DATA_BLOCK "TRAVEL_PROFIBUS"	// DB 18
VERSION : 0.1
  STRUCT
   TRVLDRV1_REF_WITH_LIMIT : BOOL ;	//TRAVEL DRIVE-1 RESERVED1 BIT
   TRVLDRV1_LOCAL_REMOTE_BI : BOOL ;	//TRAVEL DRIVE-1 PROFIBUS SELECTED BIT
   TRVLDRV1_ACT_ABOVE_LMIT : BOOL ;	//TRAVEL DRIVE-1 REFERENCE REACHED BIT
   TRVLDRV1_PROFI_SELECTED : BOOL ;	//TRAVEL DRIVE-1 RESERVED2 BIT
   TRVLDRV1_EXTRNL_RUN_BIT : BOOL ;	//TRAVEL DRIVE-1 RESERVED3 BIT
   TRVLDRV1_RESERVED1_BIT : BOOL ;	//TRAVEL DRIVE-1 RESERVED4 BIT
   TRVLDRV1_RESERVED2_BIT : BOOL ;	//TRAVEL DRIVE-1 RESERVED5 BIT
   TRVLDRV1_RESERVED3_BIT : BOOL ;	//TRAVEL DRIVE-1 REVERSE DIRECTION BIT
   TRVLDRV1_RDY_SWITCH_ON : BOOL ;	//TRAVEL DRIVE-1 READY TO SWITCH ON BIT
   TRVLDRV1_RDY_BIT : BOOL ;	//TRAVEL DRIVE-1 READY BIT
   TRVLDRV1_RUNNING_BIT : BOOL ;	//TRAVEL DRIVE-1 RUNNING BIT
   TRVLDRV1_FAULT_BIT : BOOL ;	//TRAVEL DRIVE-1 FAULT BIT
   TRVLDRV1_OFF2_BIT : BOOL ;	//TRAVEL DRIVE-1 VOLTAGE ENABLED BIT
   TRVLDRV1_OFF3_BIT : BOOL ;	//TRAVEL DRIVE-1 EMERGENCY STOP BIT
   TRVLDRV1_SWTCHON_DISABLE : BOOL ;	//TRAVEL DRIVE-1 SWITCH ON DISABLE BIT
   TRVLDRV1_ALARM_BIT : BOOL ;	//TRAVEL DRIVE-1 ALARM BIT
   TRVLDRV1_SPEED_ACTUAL : INT ;	//TRAVEL DRIVE-1 SPEED ACTUAL VALUE
   TRAV_DRV_1_CURR_VAL : INT ;	//TRAVEL DRIVE 1 CURRENT VALUE
   TRV1_SPARE2_STATUS : WORD ;	//Temporary placeholder variable
   TRV1_SPARE3_STATUS : WORD ;	//Temporary placeholder variable
   TRV1_SPARE4_STATUS : WORD ;	//Temporary placeholder variable
   TRV1_SPARE5_STATUS : WORD ;	//Temporary placeholder variable
   TRV1_SPARE6_STATUS : WORD ;	//Temporary placeholder variable
   TRV1_SPARE7_STATUS : WORD ;	//Temporary placeholder variable
   TRV1_SPARE8_STATUS : WORD ;	//Temporary placeholder variable
   TRVLDRV1_CONTROLWORD : WORD ;	//TRAVEL DRIVE-1 CONTROL WORD VALUE
   TRVLDRV1_SPEED_REF : INT ;	//TRVVEL DRIVE-1 SPEED REFERENCE VALUE
   PZD3_DW1_3 : WORD ;	//PROCESS DATA FOR DRIVE
   TRV1_SPARE2_CNTL_WORD : WORD ;	//Temporary placeholder variable
   TRV1_SPARE3_CNTL_WORD : WORD ;	//Temporary placeholder variable
   TRV1_SPARE4_CNTL_WORD : WORD ;	//Temporary placeholder variable
   TRV1_SPARE5_CNTL_WORD : WORD ;	//Temporary placeholder variable
   TRV1_SPARE6_CNTL_WORD : WORD ;	//Temporary placeholder variable
   TRV1_SPARE7_CNTL_WORD : WORD ;	//Temporary placeholder variable
   TRV1_SPARE8_CNTL_WORD : WORD ;	//Temporary placeholder variable
   TRVLDRV2_REF_WITH_LIMIT : BOOL ;	//TRAVEL DRIVE-2 RESERVED1 BIT
   TRVLDRV2_LOCAL_REMOTE_BI : BOOL ;	//TRAVEL DRIVE-2 PROFIBUS SELECTED BIT
   TRVLDRV2_ACT_ABOVE_LMIT : BOOL ;	//TRAVEL DRIVE-2 REFERENCE REACHED BIT
   TRVLDRV2_PROFI_SELECTED : BOOL ;	//TRAVEL DRIVE-2 RESERVED2 BIT
   TRVLDRV2_EXTRNL_RUN_BIT : BOOL ;	//TRAVEL DRIVE-2 RESERVED3 BIT
   TRVLDRV2_RESERVED1_BIT : BOOL ;	//TRAVEL DRIVE-2 RESERVED4 BIT
   TRVLDRV2_RESERVED2_BIT : BOOL ;	//TRAVEL DRIVE-2 RESERVED5 BIT
   TRVLDRV2_RESERVED3_BIT : BOOL ;	//TRAVEL DRIVE-2 REVERSE DIRECTION BIT
   TRVLDRV2_RDY_SWITCH_ON : BOOL ;	//TRAVEL DRIVE-2 READY TO SWITCH ON BIT
   TRVLDRV2_RDY_BIT : BOOL ;	//TRAVEL DRIVE-2 READY BIT
   TRVLDRV2_RUNNING_BIT : BOOL ;	//TRAVEL DRIVE-2 RUNNING BIT
   TRVLDRV2_FAULT_BIT : BOOL ;	//TRAVEL DRIVE-2 FAULT BIT
   TRVLDRV2_OFF2_BIT : BOOL ;	//TRAVEL DRIVE-2 VOLTAGE ENABLED BIT
   TRVLDRV2_OFF3_BIT : BOOL ;	//TRAVEL DRIVE-2 EMERGENCY STOP BIT
   STAT_2 : BOOL ;	//TRAVEL DRIVE-2 SWITCH ON DISABLE BIT
   TRVLDRV2_ALARM_BIT : BOOL ;	//TRAVEL DRIVE-2 ALARM BIT
   TRVLDRV2_SPEED_ACTUAL : INT ;	//TRAVEL DRIVE-2 SPEED ACTUAL VALUE
   TRAV_DRV_2_CURR_VAL : INT ;	//TRAVEL DRIVE 2 CURRENT VALUE
   TRV2_SPARE2_STATUS : WORD ;	//Temporary placeholder variable
   TRV2_SPARE3_STATUS : WORD ;	//Temporary placeholder variable
   TRV2_SPARE4_STATUS : WORD ;	//Temporary placeholder variable
   TRV2_SPARE5_STATUS : WORD ;	//Temporary placeholder variable
   TRV2_SPARE6_STATUS : WORD ;	//Temporary placeholder variable
   TRV2_SPARE7_STATUS : WORD ;	//Temporary placeholder variable
   TRV2_SPARE8_STATUS : WORD ;	//Temporary placeholder variable
   TRVLDRV2_CONTROLWORD : WORD ;	//TRAVEL DRIVE-2 CONTROL WORD VALUE
   TRVLDRV2_SPEED_REF : INT ;	//TRVVEL DRIVE-2 SPEED REFERENCE VALUE
   TRVLDRV2_REF_2 : WORD ;	//TRAVEL DRIVE-2 SPEED REFERENCE VALUE
   AUX_DS_REF3 : WORD ;	//AUXILLIARY DATA SET REF 3
   TRV2_SPARE3_CNTL_WORD : WORD ;	//Temporary placeholder variable
   TRV2_SPARE4_CNTL_WORD : WORD ;	//Temporary placeholder variable
   TRV2_SPARE5_CNTL_WORD : WORD ;	//Temporary placeholder variable
   TRV2_SPARE6_CNTL_WORD : WORD ;	//Temporary placeholder variable
   TRV2_SPARE7_CNTL_WORD : WORD ;	//Temporary placeholder variable
   TRV2_SPARE8_CNTL_WORD : WORD ;	//Temporary placeholder variable
  END_STRUCT ;	
BEGIN
END_DATA_BLOCK

DATA_BLOCK "SF_PROFIBUS"	// DB 19
VERSION : 0.1
  STRUCT
   SF1_REF_WITH_LIMIT : BOOL ;	//SCREW FEEDER DRIVE-1 RESERVED1 BIT
   SF1_LOCAL_REMOTE_BI : BOOL ;	//SCREW FEEDER DRIVE-1 PROFIBUS SELECTED BIT
   SF1_ACT_ABOVE_LMIT : BOOL ;	//SCREW FEEDER DRIVE-1 REFERENCE REACHED BIT
   SF1_PROFI_SELECTED : BOOL ;	//SCREW FEEDER DRIVE-1 RESERVED2 BIT
   SF1_EXTRNL_RUN_BIT : BOOL ;	//SCREW FEEDER DRIVE-1 RESERVED3 BIT
   SF1_RESERVED1_BIT : BOOL ;	//SCREW FEEDER DRIVE-1 RESERVED4 BIT
   SF1_RESERVED2_BIT : BOOL ;	//SCREW FEEDER DRIVE-1 RESERVED5 BIT
   SF1_RESERVED3_BIT : BOOL ;	//SCREW FEEDER DRIVE-1 REVERSE DIRECTION BIT
   SF1_RDY_SWITCH_ON : BOOL ;	//SCREW FEEDER DRIVE-1 READY TO SWITCH ON BIT
   SF1_RDY_BIT : BOOL ;	//SCREW FEEDER DRIVE-1 READY BIT
   SF1_RUNNING_BIT : BOOL ;	//SCREW FEEDER DRIVE-1 RUNNING BIT
   SF1_FAULT_BIT : BOOL ;	//SCREW FEEDER DRIVE-1 FAULT BIT
   SF1_OFF2_BIT : BOOL ;	//SCREW FEEDER DRIVE-1 VOLTAGE ENABLED BIT
   SF1_OFF3_BIT : BOOL ;	//SCREW FEEDER DRIVE-1 EMERGENCY STOP BIT
   SF1_SWTCHON_DISABLE : BOOL ;	//SCREW FEEDER DRIVE-1 SWITCH ON DISABLE BIT
   SF1_ALARM_BIT : BOOL ;	//SCREW FEEDER DRIVE-1 ALARM BIT
   SF1_SPEED_ACTUAL : INT ;	//SCREW FEEDER DRIVE-1 SPEED ACTUAL VALUE
   SF_1_CURR_VAL : INT ;	//SCREW FEEDER DRIVE-1 CURRENT VALUE
   SF1_SPARE2_STATUS : WORD ;	//SCREW FEEDER SPARE STATUS WORD
   SF1_SPARE3_STATUS : WORD ;	//SCREW FEEDER SPARE STATUS WORD
   SF1_SPARE4_STATUS : WORD ;	//SCREW FEEDER SPARE STATUS WORD
   SF1_SPARE5_STATUS : WORD ;	//SCREW FEEDER SPARE STATUS WORD
   SF1_SPARE6_STATUS : WORD ;	//SCREW FEEDER SPARE STATUS WORD
   SF1_SPARE7_STATUS : WORD ;	//SCREW FEEDER SPARE STATUS WORD
   SF1_SPARE8_STATUS : WORD ;	//SCREW FEEDER SPARE STATUS WORD
   SF1_CONTROLWORD : WORD ;	//SCREW FEEDER DRIVE-1 CONTROL WORD VALUE
   SF1_SPEED_REF : INT ;	//SCREW FEEDER DRIVE-1 SPEED REFERENCE VALUE
   SF1_SPARE1_CNTL_WORD : WORD ;	//SCREW FEEDER SPARE CONTROL WORD
   SF1_SPARE2_CNTL_WORD : WORD ;	//SCREW FEEDER SPARE CONTROL WORD
   SF1_SPARE3_CNTL_WORD : WORD ;	//SCREW FEEDER SPARE CONTROL WORD
   SF1_SPARE4_CNTL_WORD : WORD ;	//SCREW FEEDER SPARE CONTROL WORD
   SF1_SPARE5_CNTL_WORD : WORD ;	//SCREW FEEDER SPARE CONTROL WORD
   SF1_SPARE6_CNTL_WORD : WORD ;	//SCREW FEEDER SPARE CONTROL WORD
   SF1_SPARE7_CNTL_WORD : WORD ;	//SCREW FEEDER SPARE CONTROL WORD
   SF1_SPARE8_CNTL_WORD : WORD ;	//SCREW FEEDER SPARE CONTROL WORD
   SF2_REF_WITH_LIMIT : BOOL ;	//SCREW FEEDER DRIVE-2 RESERVED1 BIT
   SF2_LOCAL_REMOTE_BIT : BOOL ;	//SCREW FEEDER DRIVE-2 PROFIBUS SELECTED BIT
   SF2_ACT_ABOVE_LMIT : BOOL ;	//SCREW FEEDER DRIVE-2 REFERENCE REACHED BIT
   SF2_PROFI_SELECTED : BOOL ;	//SCREW FEEDER DRIVE-2 RESERVED2 BIT
   SF2_EXTRNL_RUN_BIT : BOOL ;	//SCREW FEEDER DRIVE-2 RESERVED3 BIT
   SF2_RESERVED1_BIT1 : BOOL ;	//SCREW FEEDER DRIVE-2 RESERVED4 BIT
   SF2_RESERVED2_BIT : BOOL ;	//SCREW FEEDER DRIVE-2 RESERVED5 BIT
   SF2_RESERVED3_BIT : BOOL ;	//SCREW FEEDER DRIVE-2 REVERSE DIRECTION BIT
   SF2_RDY_SWITCH_ON : BOOL ;	//SCREW FEEDER DRIVE-2 READY TO SWITCH ON BIT
   SF2_RDY_BIT : BOOL ;	//SCREW FEEDER DRIVE-2 READY BIT
   SF2_RUNNING_BIT : BOOL ;	//SCREW FEEDER DRIVE-2 RUNNING BIT
   SF2_FAULT_BIT : BOOL ;	//SCREW FEEDER DRIVE-2 FAULT BIT
   SF2_OFF2_BIT : BOOL ;	//SCREW FEEDER DRIVE-2 VOLTAGE ENABLED BIT
   SF2_OFF3_BIT : BOOL ;	//SCREW FEEDER DRIVE-2 EMERGENCY STOP BIT
   SF2_SWTCHON_DISABLE : BOOL ;	//SCREW FEEDER DRIVE-2 SWITCH ON DISABLE BIT
   SF2_ALARM_BIT : BOOL ;	//SCREW FEEDER DRIVE-2 ALARM BIT
   SF2_SPEED_ACTUAL : INT ;	//SCREW FEEDER DRIVE-2 SPEED ACTUAL VALUE
   SF_2_CURR_VAL : INT ;	//SCREW FEEDER DRIVE 2 CURRENT VALUE
   SF2_SPARE2_STATUS : WORD ;	//SCREW FEEDER SPARE STATUS WORD
   SF2_SPARE3_STATUS : WORD ;	//SCREW FEEDER SPARE STATUS WORD
   SF2_SPARE4_STATUS : WORD ;	//SCREW FEEDER SPARE STATUS WORD
   SF2_SPARE5_STATUS : WORD ;	//SCREW FEEDER SPARE STATUS WORD
   SF2_SPARE6_STATUS : WORD ;	//SCREW FEEDER SPARE STATUS WORD
   SF2_SPARE7_STATUS : WORD ;	//SCREW FEEDER SPARE STATUS WORD
   SF2_SPARE8_STATUS : WORD ;	//SCREW FEEDER SPARE STATUS WORD
   SF2_CONTROLWORD : WORD ;	//SCREW FEEDER DRIVE-2 CONTROL WORD VALUE
   SF2_SPEED_REF : INT ;	//SCREW FEEDER DRIVE-2 SPEED REFERENCE VALUE
   SF2_SPARE1_CNTL_WORD : WORD ;	//SCREW FEEDER SPARE CONTROL WORD
   SF2_SPARE2_CNTL_WORD : WORD ;	//SCREW FEEDER SPARE CONTROL WORD
   SF2_SPARE3_CNTL_WORD : WORD ;	//SCREW FEEDER SPARE CONTROL WORD
   SF2_SPARE4_CNTL_WORD : WORD ;	//SCREW FEEDER SPARE CONTROL WORD
   SF2_SPARE5_CNTL_WORD : WORD ;	//SCREW FEEDER SPARE CONTROL WORD
   SF2_SPARE6_CNTL_WORD : WORD ;	//SCREW FEEDER SPARE CONTROL WORD
   SF2_SPARE7_CNTL_WORD : WORD ;	//SCREW FEEDER SPARE CONTROL WORD
   SF2_SPARE8_CNTL_WORD : WORD ;	//SCREW FEEDER SPARE CONTROL WORD
   SF3_REF_WITH_LIMIT : BOOL ;	//SCREW FEEDER DRIVE-3 RESERVED1 BIT
   SF3_LOCAL_REMOTE_BIT : BOOL ;	//SCREW FEEDER DRIVE-3 PROFIBUS SELECTED BIT
   SF3_ACT_ABOVE_LMIT : BOOL ;	//SCREW FEEDER DRIVE-3 REFERENCE REACHED BIT
   SF3_PROFI_SELECTED : BOOL ;	//SCREW FEEDER DRIVE-3 RESERVED2 BIT
   SF3_EXTRNL_RUN_BIT : BOOL ;	//SCREW FEEDER DRIVE-3 RESERVED3 BIT
   SF3_RESERVED1_BIT : BOOL ;	//SCREW FEEDER DRIVE-3 RESERVED4 BIT
   SF3_RESERVED2_BIT : BOOL ;	//SCREW FEEDER DRIVE-3 RESERVED5 BIT
   SF3_RESERVED3_BIT : BOOL ;	//SCREW FEEDER DRIVE-3 REVERSE DIRECTION BIT
   SF3_RDY_SWITCH_ON : BOOL ;	//SCREW FEEDER DRIVE-3 READY TO SWITCH ON BIT
   SF3_RDY_BIT : BOOL ;	//SCREW FEEDER DRIVE-3 READY BIT
   SF3_RUNNING_BIT : BOOL ;	//SCREW FEEDER DRIVE-3 RUNNING BIT
   SF3_FAULT_BIT : BOOL ;	//SCREW FEEDER DRIVE-3 FAULT BIT
   SF3_OFF2_BIT : BOOL ;	//SCREW FEEDER DRIVE-3 VOLTAGE ENABLED BIT
   SF3_OFF3_BIT : BOOL ;	//SCREW FEEDER DRIVE-3 EMERGENCY STOP BIT
   SF3_SWTCHON_DISABLE : BOOL ;	//SCREW FEEDER DRIVE-3 SWITCH ON DISABLE BIT
   SF3_ALARM_BIT : BOOL ;	//SCREW FEEDER DRIVE-3 ALARM BIT
   SF3_SPEED_ACTUAL : INT ;	//SCREW FEEDER DRIVE-3 SPEED ACTUAL VALUE
   SF_3_CURR_VAL : INT ;	//SCREW FEEDER DRIVE-3 CURRENT VALUE
   SF3_SPARE2_STATUS : WORD ;	//SCREW FEEDER SPARE STATUS WORD
   SF3_SPARE3_STATUS : WORD ;	//SCREW FEEDER SPARE STATUS WORD
   SF3_SPARE4_STATUS : WORD ;	//SCREW FEEDER SPARE STATUS WORD
   SF3_SPARE5_STATUS : WORD ;	//SCREW FEEDER SPARE STATUS WORD
   SF3_SPARE6_STATUS : WORD ;	//SCREW FEEDER SPARE STATUS WORD
   SF3_SPARE7_STATUS : WORD ;	//SCREW FEEDER SPARE STATUS WORD
   SF3_SPARE8_STATUS : WORD ;	//SCREW FEEDER SPARE STATUS WORD
   SF3_CONTROLWORD : WORD ;	//SCREW FEEDER DRIVE-3 CONTROL WORD VALUE
   SF3_SPEED_REF : INT ;	//SCREW FEEDER DRIVE-3 SPEED REFERENCE VALUE
   SF3_SPARE1_CNTL_WORD : WORD ;	//SCREW FEEDER SPARE CONTROL WORD
   SF3_SPARE2_CNTL_WORD : WORD ;	//SCREW FEEDER SPARE CONTROL WORD
   SF3_SPARE3_CNTL_WORD : WORD ;	//SCREW FEEDER SPARE CONTROL WORD
   SF3_SPARE4_CNTL_WORD : WORD ;	//SCREW FEEDER SPARE CONTROL WORD
   SF3_SPARE5_CNTL_WORD : WORD ;	//SCREW FEEDER SPARE CONTROL WORD
   SF3_SPARE6_CNTL_WORD : WORD ;	//SCREW FEEDER SPARE CONTROL WORD
   SF3_SPARE7_CNTL_WORD : WORD ;	//SCREW FEEDER SPARE CONTROL WORD
   SF3_SPARE8_CNTL_WORD : WORD ;	//SCREW FEEDER SPARE CONTROL WORD
  END_STRUCT ;	
BEGIN
END_DATA_BLOCK

ORGANIZATION_BLOCK "MAIN_PROGRAM"	// OB 1
TITLE = "Main Program Sweep (Cycle)"
AUTHOR : Arun_Ram
VERSION : 0.1
VAR_TEMP
  OB1_EV_CLASS : BYTE ;	//Bits 0-3 = 1 (Coming event), Bits 4-7 = 1 (Event class 1)
  OB1_SCAN_1 : BYTE ;	//1 (Cold restart scan 1 of OB 1), 3 (Scan 2-n of OB 1)
  OB1_PRIORITY : BYTE ;	//Priority of OB Execution
  OB1_OB_NUMBR : BYTE ;	//1 (Organization block 1, OB1)
  OB1_RESERVED_1 : BYTE ;	//Reserved for system
  OB1_RESERVED_2 : BYTE ;	//Reserved for system
  OB1_PREV_CYCLE : INT ;	//Cycle time of previous OB1 scan (milliseconds)
  OB1_MIN_CYCLE : INT ;	//Minimum cycle time of OB1 (milliseconds)
  OB1_MAX_CYCLE : INT ;	//Maximum cycle time of OB1 (milliseconds)
  OB1_DATE_TIME : DATE_AND_TIME ;	//Date and time OB1 started
  temp1 : INT ;
END_VAR
BEGIN
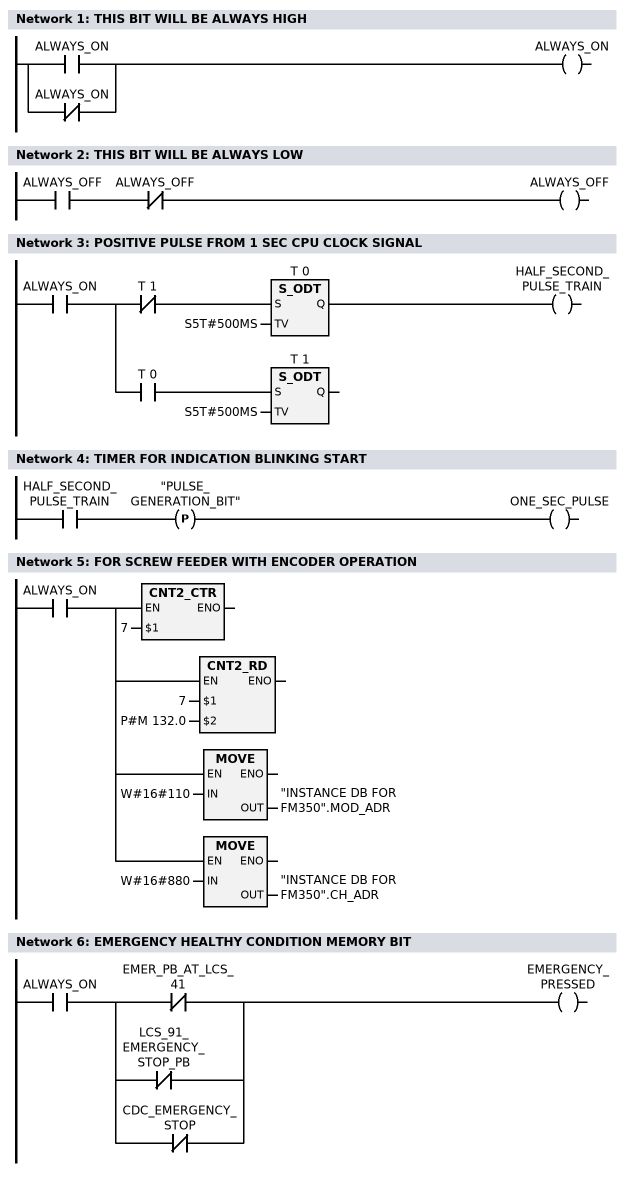
NETWORK
TITLE = THIS BIT WILL BE ALWAYS HIGH
//this bit will be always high
//TESTING PURPOSE M 0.1 THIS BIT IS ALWAYS HIGH
      O     "ALWAYS_ON";
      ON    "ALWAYS_ON";
      =     "ALWAYS_ON";
NETWORK
TITLE = THIS BIT WILL BE ALWAYS LOW
//this bit will be always low
//TESTING PURPOSE M 0.0 THIS BIT IS ALWAYS LOW
      A     "ALWAYS_OFF";
      AN    "ALWAYS_OFF";
      =     "ALWAYS_OFF";
NETWORK
TITLE = POSITIVE PULSE FROM 1 SEC CPU CLOCK SIGNAL
      A     "ALWAYS_ON";
      =     L 22.0;
      A     L 22.0;
      AN    T 1;
      L     S5T#500MS;
      SD    T 0;
      NOP   0;
      NOP   0;
      NOP   0;
      A     T 0;
      =     "HALF_SECOND_PULSE_TRAIN";
      A     L 22.0;
      A     T 0;
      L     S5T#500MS;
      SD    T 1;
      NOP   0;
      NOP   0;
      NOP   0;
      NOP   0;
NETWORK
TITLE = TIMER FOR INDICATION BLINKING START
//T5 TIMER WILL GIVE BLINKING PULSES FOR INDICATION LAMPS
      A     "HALF_SECOND_PULSE_TRAIN";
      FP    "PULSE_GENERATION_BIT";
      =     "ONE_SEC_PULSE";
NETWORK
TITLE = FOR SCREW FEEDER WITH ENCODER OPERATION
//CALLING THE OPERATION SEQUENCE BLOCK FOR FUNCTION MODULE FM 350-2
      A     "ALWAYS_ON";
      =     L 22.0;
      A     L 22.0;
      JNB   _001;
      CALL  "CNT2_CTR" (
           $1                       := 7);
_001: NOP   0;
      A     L 22.0;
      JNB   _002;
      CALL  "CNT2_RD" (
           $1                       := 7,
           $2                       := P#M 132.0);
_002: NOP   0;
      A     L 22.0;
      JNB   _003;
      L     W#16#110;
      T     "INSTANCE DB FOR FM350".MOD_ADR;
_003: NOP   0;
      A     L 22.0;
      JNB   _004;
      L     W#16#880;
      T     "INSTANCE DB FOR FM350".CH_ADR;
_004: NOP   0;
NETWORK
TITLE = EMERGENCY HEALTHY CONDITION MEMORY BIT
//this emergency bit is used to block all the outputs
//M 11.7 WILL BE NOT ASSIGNED IF ALL THE EMERGENCY PB ARE HEALTHY CONDITION
      A     "ALWAYS_ON";
      A(;
      ON    "EMER_PB_AT_LCS_41";
      ON    "LCS_91_EMERGENCY_STOP_PB";
      ON    "CDC_EMERGENCY_STOP";
      );
      =     "EMERGENCY_PRESSED";
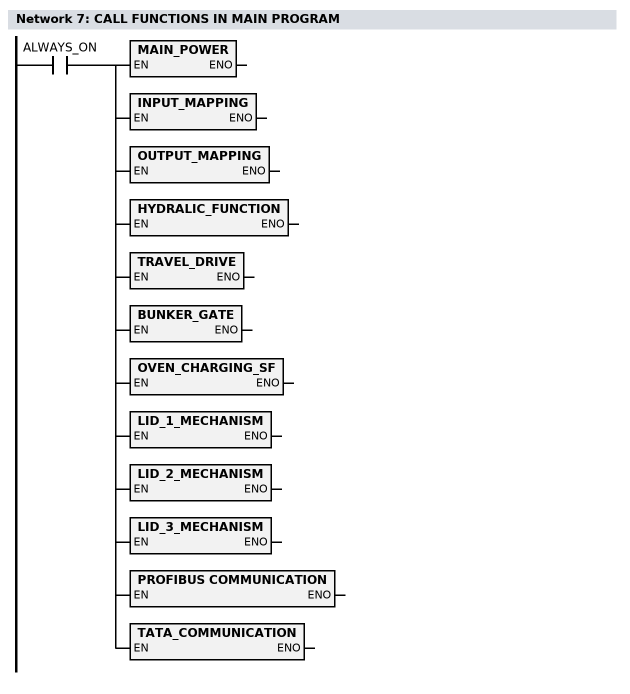
NETWORK
TITLE = CALL FUNCTIONS IN MAIN PROGRAM
      A     "ALWAYS_ON";
      =     L 22.0;
      A     L 22.0;
      JNB   _005;
      CALL  "MAIN_POWER";
_005: NOP   0;
      A     L 22.0;
      JNB   _006;
      CALL  "INPUT_MAPPING";
_006: NOP   0;
      A     L 22.0;
      JNB   _007;
      CALL  "OUTPUT_MAPPING";
_007: NOP   0;
      A     L 22.0;
      JNB   _008;
      CALL  "HYDRALIC_FUNCTION";
_008: NOP   0;
      A     L 22.0;
      JNB   _009;
      CALL  "TRAVEL_DRIVE";
_009: NOP   0;
      A     L 22.0;
      JNB   _00a;
      CALL  "BUNKER_GATE";
_00a: NOP   0;
      A     L 22.0;
      JNB   _00b;
      CALL  "OVEN_CHARGING_SF";
_00b: NOP   0;
      A     L 22.0;
      JNB   _00c;
      CALL  "LID_1_MECHANISM";
_00c: NOP   0;
      A     L 22.0;
      JNB   _00d;
      CALL  "LID_2_MECHANISM";
_00d: NOP   0;
      A     L 22.0;
      JNB   _00e;
      CALL  "LID_3_MECHANISM";
_00e: NOP   0;
      A     L 22.0;
      JNB   _00f;
      CALL  "PROFIBUS COMMUNICATION";
_00f: NOP   0;
      A     L 22.0;
      JNB   _010;
      CALL  "TATA_COMMUNICATION";
_010: NOP   0;
END_ORGANIZATION_BLOCK

ORGANIZATION_BLOCK "CYCL_FLT"	// OB 80
TITLE = "Cycle Time Fault"
VERSION : 0.1
VAR_TEMP
  OB80_EV_CLASS : BYTE ;	//16#35, Event class 3, Entering event state, Internal fault event
  OB80_FLT_ID : BYTE ;	//16#XX, Fault identifcation code
  OB80_PRIORITY : BYTE ;	//Priority of OB Execution
  OB80_OB_NUMBR : BYTE ;	//80 (Organization block 80, OB80)
  OB80_RESERVED_1 : BYTE ;	//Reserved for system
  OB80_RESERVED_2 : BYTE ;	//Reserved for system
  OB80_ERROR_INFO : WORD ;	//Error information on event
  OB80_ERR_EV_CLASS : BYTE ;	//Class of event causing error
  OB80_ERR_EV_NUM : BYTE ;	//Number of event causing error
  OB80_OB_PRIORITY : BYTE ;	//Priority of OB causing error
  OB80_OB_NUM : BYTE ;	//Number of OB causing error
  OB80_DATE_TIME : DATE_AND_TIME ;	//Date and time OB80 started
END_VAR
BEGIN
// (block stored without names or comments; labels and parameter names are numbered)
END_ORGANIZATION_BLOCK

ORGANIZATION_BLOCK "I/O_FLT1"	// OB 82
TITLE = "I/O Point Fault"
VERSION : 0.1
VAR_TEMP
  OB82_EV_CLASS : BYTE ;	//16#39, Event class 3, Entering event state, Internal fault event
  OB82_FLT_ID : BYTE ;	//16#XX, Fault identifcation code
  OB82_PRIORITY : BYTE ;	//Priority of OB Execution
  OB82_OB_NUMBR : BYTE ;	//82 (Organization block 82, OB82)
  OB82_RESERVED_1 : BYTE ;	//Reserved for system
  OB82_IO_FLAG : BYTE ;	//Input (01010100), Output (01010101)
  OB82_MDL_ADDR : WORD ;	//Base address of module with fault
  OB82_MDL_DEFECT : BOOL ;	//Module defective
  OB82_INT_FAULT : BOOL ;	//Internal fault
  OB82_EXT_FAULT : BOOL ;	//External fault
  OB82_PNT_INFO : BOOL ;	//Point information
  OB82_EXT_VOLTAGE : BOOL ;	//External voltage low
  OB82_FLD_CONNCTR : BOOL ;	//Field wiring connector missing
  OB82_NO_CONFIG : BOOL ;	//Module has no configuration data
  OB82_CONFIG_ERR : BOOL ;	//Module has configuration error
  OB82_MDL_TYPE : BYTE ;	//Type of module
  OB82_SUB_MDL_ERR : BOOL ;	//Sub-Module is missing or has error
  OB82_COMM_FAULT : BOOL ;	//Communication fault
  OB82_MDL_STOP : BOOL ;	//Module is stopped
  OB82_WTCH_DOG_FLT : BOOL ;	//Watch dog timer stopped module
  OB82_INT_PS_FLT : BOOL ;	//Internal power supply fault
  OB82_PRIM_BATT_FLT : BOOL ;	//Primary battery is in fault
  OB82_BCKUP_BATT_FLT : BOOL ;	//Backup battery is in fault
  OB82_RESERVED_2 : BOOL ;	//Reserved for system
  OB82_RACK_FLT : BOOL ;	//Rack fault, only for bus interface module
  OB82_PROC_FLT : BOOL ;	//Processor fault
  OB82_EPROM_FLT : BOOL ;	//EPROM fault
  OB82_RAM_FLT : BOOL ;	//RAM fault
  OB82_ADU_FLT : BOOL ;	//ADU fault
  OB82_FUSE_FLT : BOOL ;	//Fuse fault
  OB82_HW_INTR_FLT : BOOL ;	//Hardware interupt input in fault
  OB82_RESERVED_3 : BOOL ;	//Reserved for system
  OB82_DATE_TIME : DATE_AND_TIME ;	//Date and time OB82 started
END_VAR
BEGIN
// (block stored without names or comments; labels and parameter names are numbered)
END_ORGANIZATION_BLOCK

ORGANIZATION_BLOCK "OBNL_FLT"	// OB 85
TITLE = "Organization Block (OB) Not Loaded Fault"
VERSION : 0.1
VAR_TEMP
  OB85_EV_CLASS : BYTE ;	//16#35 Event class 3
  OB85_FLT_ID : BYTE ;	//16#XX, Fault identification code
  OB85_PRIORITY : BYTE ;	//Priority of OB Execution
  OB85_OB_NUMBR : BYTE ;	//85 (Organization block 85, OB85)
  OB85_RESERVED_1 : BYTE ;	//Reserved for system
  OB85_RESERVED_2 : BYTE ;	//Reserved for system
  OB85_RESERVED_3 : INT ;	//Reserved for system
  OB85_ERR_EV_CLASS : BYTE ;	//Class of event causing error
  OB85_ERR_EV_NUM : BYTE ;	//Number of event causing error
  OB85_OB_PRIOR : BYTE ;	//Priority of OB causing error
  OB85_OB_NUM : BYTE ;	//Number of OB causing error
  OB85_DATE_TIME : DATE_AND_TIME ;	//Date and time OB85 started
END_VAR
BEGIN
// (block stored without names or comments; labels and parameter names are numbered)
END_ORGANIZATION_BLOCK

ORGANIZATION_BLOCK "RACK_FLT"	// OB 86
TITLE = "Loss Of Rack Fault"
VERSION : 0.1
VAR_TEMP
  OB86_EV_CLASS : BYTE ;	//16#38/39 Event class 3
  OB86_FLT_ID : BYTE ;	//16#C1/C4/C5, Fault identifcation code
  OB86_PRIORITY : BYTE ;	//Priority of OB Execution
  OB86_OB_NUMBR : BYTE ;	//86 (Organization block 86, OB86)
  OB86_RESERVED_1 : BYTE ;	//Reserved for system
  OB86_RESERVED_2 : BYTE ;	//Reserved for system
  OB86_MDL_ADDR : WORD ;	//Base address of IM module in rack with fault
  OB86_RACKS_FLTD : ARRAY  [0 .. 31 ] OF BOOL ;	//Racks in fault
  OB86_DATE_TIME : DATE_AND_TIME ;	//Date and time OB86 started
END_VAR
BEGIN
// (block stored without names or comments; labels and parameter names are numbered)
END_ORGANIZATION_BLOCK

ORGANIZATION_BLOCK "COMM_FLT"	// OB 87
TITLE = "Communication Fault"
VERSION : 0.1
VAR_TEMP
  OB87_EV_CLASS : BYTE ;	//16#39 Event class 3
  OB87_FLT_ID : BYTE ;	//16#XX, Fault identifcation code
  OB87_PRIORITY : BYTE ;	//Priority of OB Execution
  OB87_OB_NUMBR : BYTE ;	//87 (Organization block 87, OB87)
  OB87_RESERVED_1 : BYTE ;	//Reserved for system
  OB87_RESERVED_2 : BYTE ;	//Reserved for system
  OB87_RESERVED_3 : WORD ;	//Reserved for system
  OB87_RESERVED_4 : DWORD ;	//Reserved for system
  OB87_DATE_TIME : DATE_AND_TIME ;	//Date and time OB87 started
END_VAR
BEGIN
// (block stored without names or comments; labels and parameter names are numbered)
END_ORGANIZATION_BLOCK

ORGANIZATION_BLOCK "COMPLETE RESTART"	// OB 100
TITLE = "Complete Restart"
VERSION : 0.1
VAR_TEMP
  OB100_EV_CLASS : BYTE ;	//16#13, Event class 1, Entering event state, Event logged in diagnostic buffer
  OB100_STRTUP : BYTE ;	//16#81/82/83/84 Method of startup
  OB100_PRIORITY : BYTE ;	//Priority of OB Execution
  OB100_OB_NUMBR : BYTE ;	//100 (Organization block 100, OB100)
  OB100_RESERVED_1 : BYTE ;	//Reserved for system
  OB100_RESERVED_2 : BYTE ;	//Reserved for system
  OB100_STOP : WORD ;	//Event that caused CPU to stop (16#4xxx)
  OB100_STRT_INFO : DWORD ;	//Information on how system started
  OB100_DATE_TIME : DATE_AND_TIME ;	//Date and time OB100 started
END_VAR
BEGIN
NETWORK
TITLE =
END_ORGANIZATION_BLOCK

ORGANIZATION_BLOCK "PROG_ERR"	// OB 121
TITLE = "Module Access Error"
VERSION : 0.1
VAR_TEMP
  OB122_EV_CLASS : BYTE ;	//16#29, Event class 2, Entering event state, Internal fault event
  OB122_SW_FLT : BYTE ;	//16#XX Software error code
  OB122_PRIORITY : BYTE ;	//Priority of OB Execution
  OB122_OB_NUMBR : BYTE ;	//122 (Organization block 122, OB122)
  OB122_BLK_TYPE : BYTE ;	//16#88/8C/8E Type of block fault occured in
  OB122_MEM_AREA : BYTE ;	//Memory area where access error occured
  OB122_MEM_ADDR : WORD ;	//Memory address where access error occured
  OB122_BLK_NUM : WORD ;	//Block number in which error occured
  OB122_PRG_ADDR : WORD ;	//Program address where error occured
  OB122_DATE_TIME : DATE_AND_TIME ;	//Date and time OB1 started
END_VAR
BEGIN
// (block stored without names or comments; labels and parameter names are numbered)
END_ORGANIZATION_BLOCK

ORGANIZATION_BLOCK "MOD_ERR"	// OB 122
TITLE = "Module Access Error"
VERSION : 0.1
VAR_TEMP
  OB122_EV_CLASS : BYTE ;	//16#29, Event class 2, Entering event state, Internal fault event
  OB122_SW_FLT : BYTE ;	//16#XX Software error code
  OB122_PRIORITY : BYTE ;	//Priority of OB Execution
  OB122_OB_NUMBR : BYTE ;	//122 (Organization block 122, OB122)
  OB122_BLK_TYPE : BYTE ;	//16#88/8C/8E Type of block fault occured in
  OB122_MEM_AREA : BYTE ;	//Memory area where access error occured
  OB122_MEM_ADDR : WORD ;	//Memory address where access error occured
  OB122_BLK_NUM : WORD ;	//Block number in which error occured
  OB122_PRG_ADDR : WORD ;	//Program address where error occured
  OB122_DATE_TIME : DATE_AND_TIME ;	//Date and time OB1 started
END_VAR
BEGIN
// (block stored without names or comments; labels and parameter names are numbered)
END_ORGANIZATION_BLOCK
